(* Logix 5000 project; controller Transcat vendor 1 type 14 code 152 rev 32.11; software revision 32.02; part 2 of 2 *)
(* tags used below, declared in another part *)
   SpeedSensorUpperHowesSpeed : REAL;
   alwaysOFF : BOOL;
   FT103 : BronkhorstFlowMeter;
   FT104 : BronkhorstFlowMeter;
   FT105 : BronkhorstFlowMeter;
   GF101 : Thayer_WB_Feeder;   // Thayer 1 Tags
   GF201 : Thayer_WB_Feeder;   // Thayer 2 Tags
   GF301 : Acrison_Feeder;   // GF103 - Small Feeder 1
   MSG_FROM_SLC500 : INT[10];
   MX101 : Howes_Mixer;
   MX201 : Howes_Mixer;
   RecipeStart : BOOL;   // Bit to start and stop a recipe execution
   UpperHowesSpeed : INT;
   VF101 : Acrison_Feeder;   // Medium Feeder Tags
   VF201 : Acrison_Feeder;   // Small Feeder 2 Tags
(* MainProgram, continued *)

ROUTINE MainRoutine   (* ladder *)
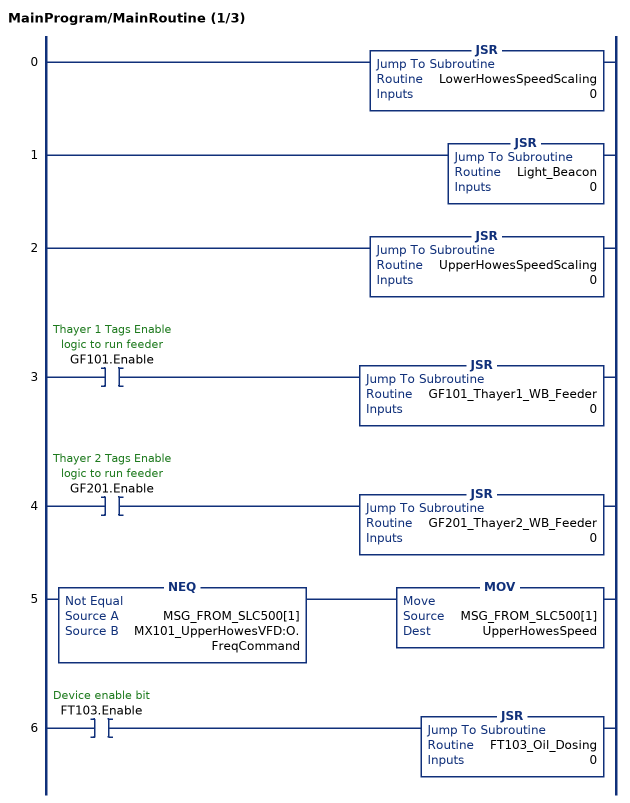
   0: JSR(LowerHowesSpeedScaling,0);
   1: JSR(Light_Beacon,0);
   2: JSR(UpperHowesSpeedScaling,0);
   3: XIC(GF101.Enable)JSR(GF101_Thayer1_WB_Feeder,0);
   4: XIC(GF201.Enable)JSR(GF201_Thayer2_WB_Feeder,0);
   5: NEQ(MSG_FROM_SLC500[1],MX101_UpperHowesVFD:O.FreqCommand)MOV(MSG_FROM_SLC500[1],UpperHowesSpeed);
   6: XIC(FT103.Enable)JSR(FT103_Oil_Dosing,0);
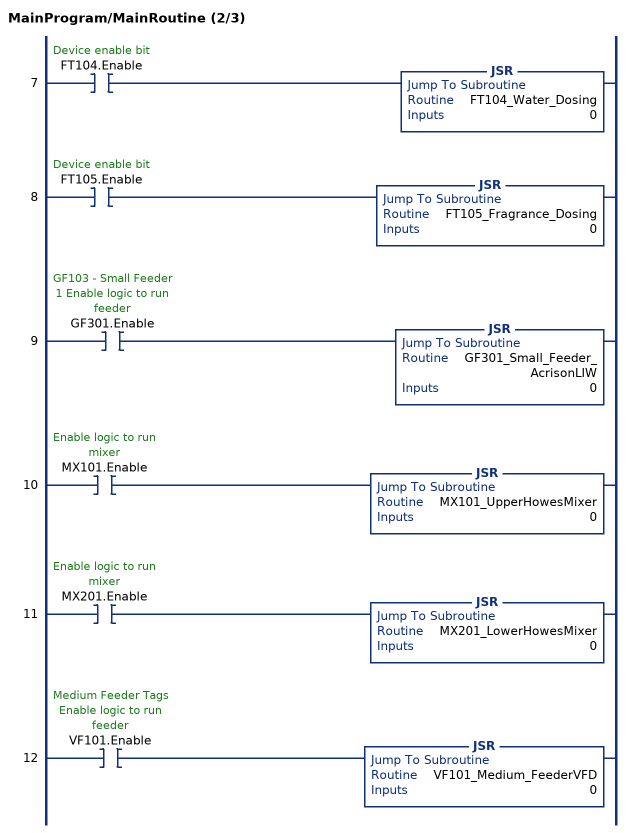
   7: XIC(FT104.Enable)JSR(FT104_Water_Dosing,0);
   8: XIC(FT105.Enable)JSR(FT105_Fragrance_Dosing,0);
   9: XIC(GF301.Enable)JSR(GF301_Small_Feeder_AcrisonLIW,0);
   10: XIC(MX101.Enable)JSR(MX101_UpperHowesMixer,0);
   11: XIC(MX201.Enable)JSR(MX201_LowerHowesMixer,0);
   12: XIC(VF101.Enable)JSR(VF101_Medium_FeederVFD,0);
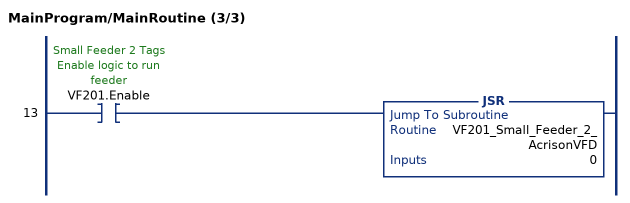
   13: XIC(VF201.Enable)JSR(VF201_Small_Feeder_2_AcrisonVFD,0);
END_ROUTINE

ROUTINE MX101_UpperHowesMixer   (* ladder *)
// Upper Howes Mixer Control Logic
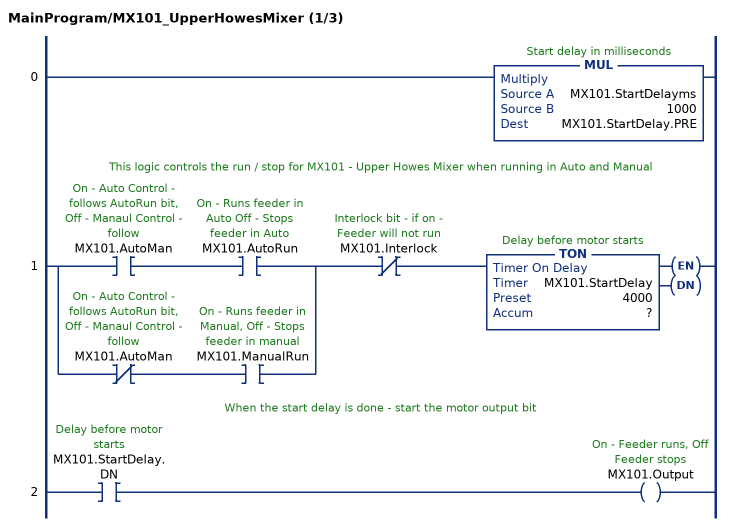
   0: MUL(MX101.StartDelayms,1000,MX101.StartDelay.PRE);
   // This logic controls the run / stop for MX101 - Upper Howes Mixer when running in Auto and Manual
   1: [XIC(MX101.AutoMan) XIC(MX101.AutoRun) ,XIO(MX101.AutoMan) XIC(MX101.ManualRun) ]XIO(MX101.Interlock)TON(MX101.StartDelay,?,?);
   // When the start delay is done - start the motor output bit
   2: XIC(MX101.StartDelay.DN)OTE(MX101.Output);
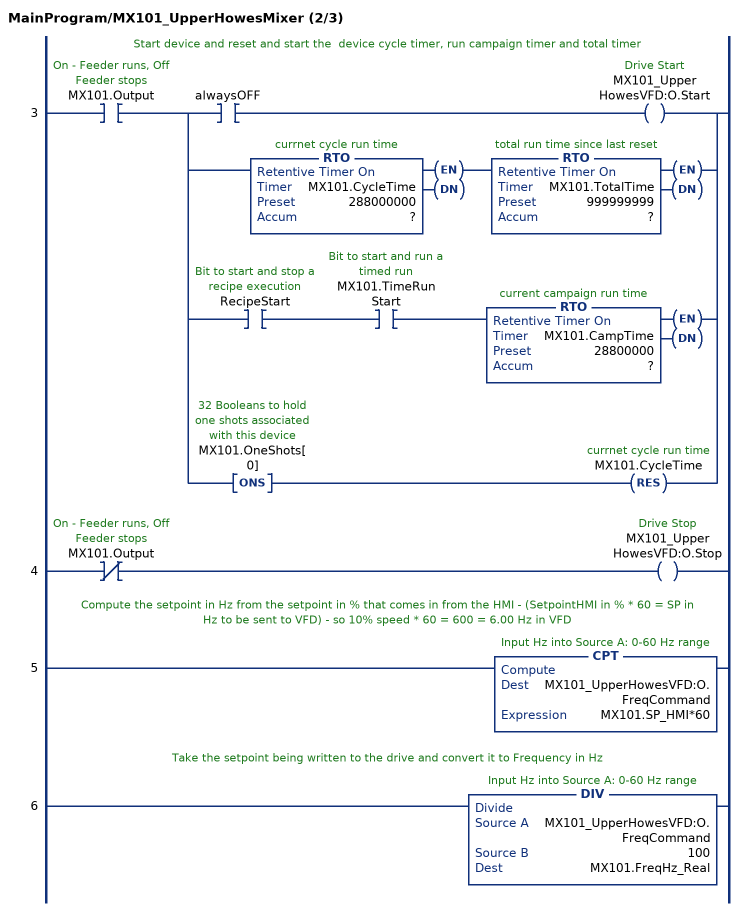
   // Start device and reset and start the  device cycle timer, run campaign timer and total timer
   3: XIC(MX101.Output)[XIC(alwaysOFF) OTE(MX101_UpperHowesVFD:O.Start) ,[RTO(MX101.CycleTime,?,?) RTO(MX101.TotalTime,?,?) ,XIC(RecipeStart) XIC(MX101.TimeRunStart) RTO(MX101.CampTime,?,?) ,ONS(MX101.OneShots[0]) RES(MX101.CycleTime) ] ];
   4: XIO(MX101.Output)OTE(MX101_UpperHowesVFD:O.Stop);
   // Compute the setpoint in Hz from the setpoint in % that comes in from the HMI - (SetpointHMI in % * 60 = SP in Hz to be sent to VFD) - so 10% speed * 60 = 600 = 6.00 Hz in VFD
   5: CPT(MX101_UpperHowesVFD:O.FreqCommand,MX101.SP_HMI*60);
   // Take the setpoint being written to the drive and convert it to Frequency in Hz
   6: DIV(MX101_UpperHowesVFD:O.FreqCommand,100,MX101.FreqHz_Real);
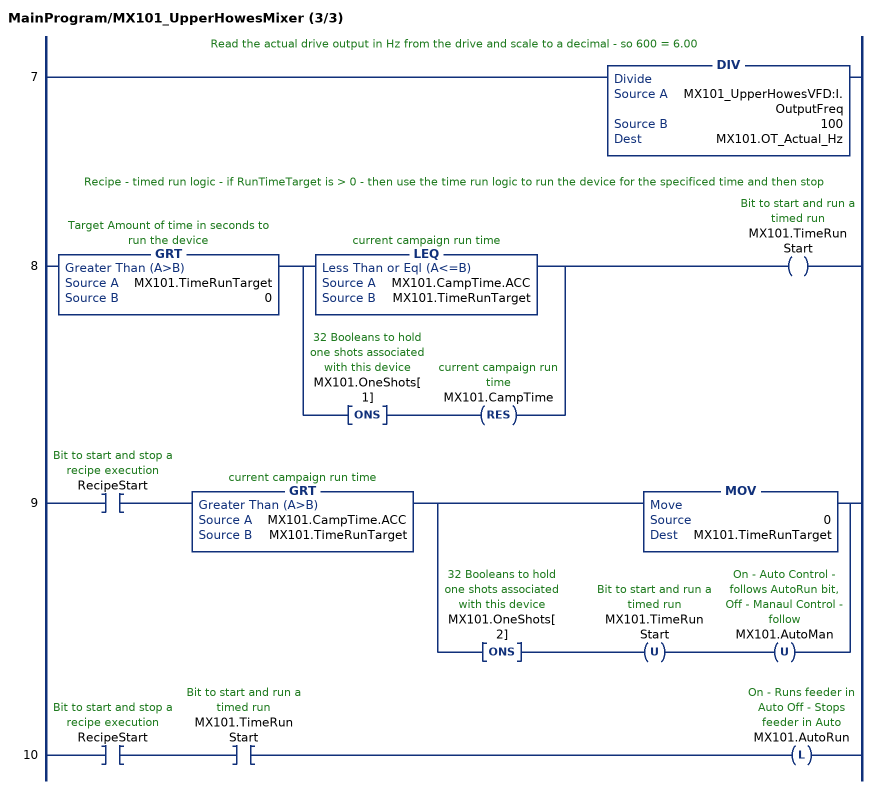
   // Read the actual drive output in Hz from the drive and scale to a decimal - so 600 = 6.00
   7: DIV(MX101_UpperHowesVFD:I.OutputFreq,100,MX101.OT_Actual_Hz);
   // Recipe - timed run logic - if RunTimeTarget is > 0 - then use the time run logic to run the device for the specificed time and then stop
   8: GRT(MX101.TimeRunTarget,0)[LEQ(MX101.CampTime.ACC,MX101.TimeRunTarget) ,ONS(MX101.OneShots[1]) RES(MX101.CampTime) ]OTE(MX101.TimeRunStart);
   9: XIC(RecipeStart)GRT(MX101.CampTime.ACC,MX101.TimeRunTarget)[MOV(0,MX101.TimeRunTarget) ,ONS(MX101.OneShots[2]) OTU(MX101.TimeRunStart) OTU(MX101.AutoMan) ];
   10: XIC(RecipeStart)XIC(MX101.TimeRunStart)OTL(MX101.AutoRun);
END_ROUTINE

ROUTINE MX201_LowerHowesMixer   (* ladder *)
// Lower Howes Mixer Control Logic
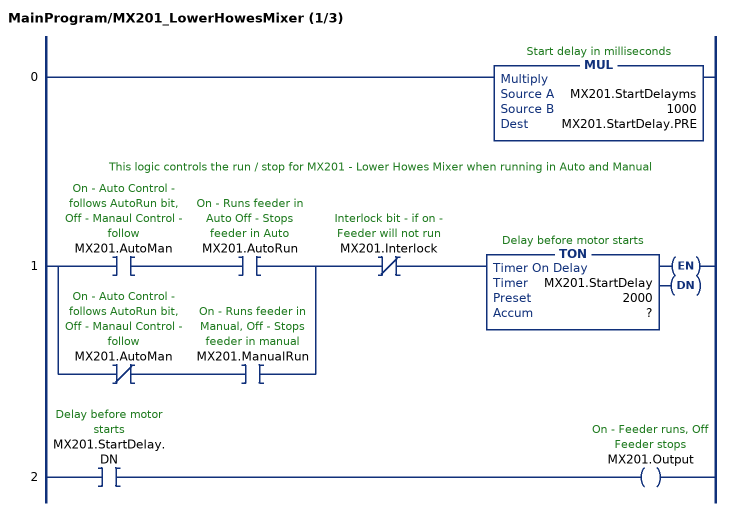
   0: MUL(MX201.StartDelayms,1000,MX201.StartDelay.PRE);
   // This logic controls the run / stop for MX201 - Lower Howes Mixer when running in Auto and Manual
   1: [XIC(MX201.AutoMan) XIC(MX201.AutoRun) ,XIO(MX201.AutoMan) XIC(MX201.ManualRun) ]XIO(MX201.Interlock)TON(MX201.StartDelay,?,?);
   2: XIC(MX201.StartDelay.DN)OTE(MX201.Output);
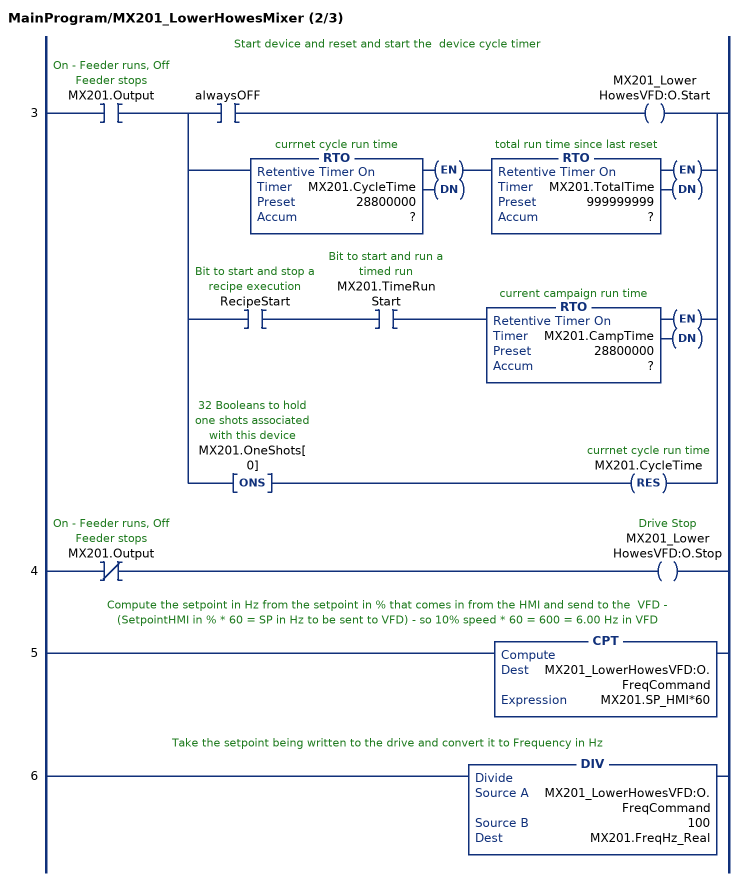
   // Start device and reset and start the  device cycle timer
   3: XIC(MX201.Output)[XIC(alwaysOFF) OTE(MX201_LowerHowesVFD:O.Start) ,[[RTO(MX201.CycleTime,?,?) RTO(MX201.TotalTime,?,?) ,XIC(RecipeStart) XIC(MX201.TimeRunStart) RTO(MX201.CampTime,?,?) ] ,ONS(MX201.OneShots[0]) RES(MX201.CycleTime) ] ];
   4: XIO(MX201.Output)OTE(MX201_LowerHowesVFD:O.Stop);
   // Compute the setpoint in Hz from the setpoint in % that comes in from the HMI and send to the  VFD - (SetpointHMI in % * 60 = SP in Hz to be sent to VFD) - so 10% speed * 60 = 600 = 6.00 Hz in VFD
   5: CPT(MX201_LowerHowesVFD:O.FreqCommand,MX201.SP_HMI*60);
   // Take the setpoint being written to the drive and convert it to Frequency in Hz
   6: DIV(MX201_LowerHowesVFD:O.FreqCommand,100,MX201.FreqHz_Real);
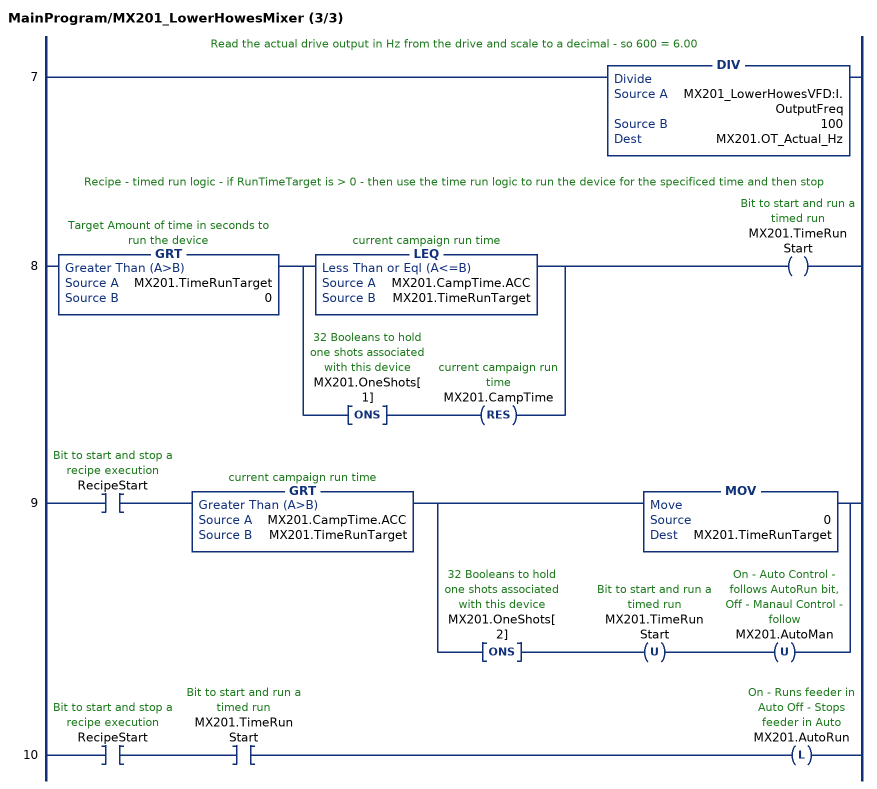
   // Read the actual drive output in Hz from the drive and scale to a decimal - so 600 = 6.00
   7: DIV(MX201_LowerHowesVFD:I.OutputFreq,100,MX201.OT_Actual_Hz);
   // Recipe - timed run logic - if RunTimeTarget is > 0 - then use the time run logic to run the device for the specificed time and then stop
   8: GRT(MX201.TimeRunTarget,0)[LEQ(MX201.CampTime.ACC,MX201.TimeRunTarget) ,ONS(MX201.OneShots[1]) RES(MX201.CampTime) ]OTE(MX201.TimeRunStart);
   9: XIC(RecipeStart)GRT(MX201.CampTime.ACC,MX201.TimeRunTarget)[MOV(0,MX201.TimeRunTarget) ,ONS(MX201.OneShots[2]) OTU(MX201.TimeRunStart) OTU(MX201.AutoMan) ];
   10: XIC(RecipeStart)XIC(MX201.TimeRunStart)OTL(MX201.AutoRun);
END_ROUTINE

ROUTINE UpperHowesSpeedScaling   (* function block diagram *)
// 4-20 MillAmp scaling
   SHEET 1
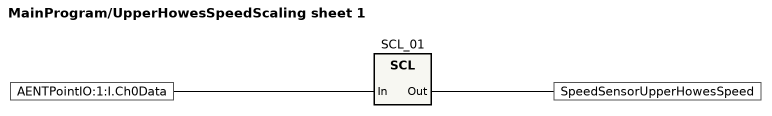
   SCL_01 : SCL(In := AENTPointIO:1:I.Ch0Data);
   SpeedSensorUpperHowesSpeed := SCL_01.Out;
END_ROUTINE

ROUTINE VF101_Medium_FeederVFD   (* ladder *)
// Medium Feeder Control via PowerFlex 525 VFD
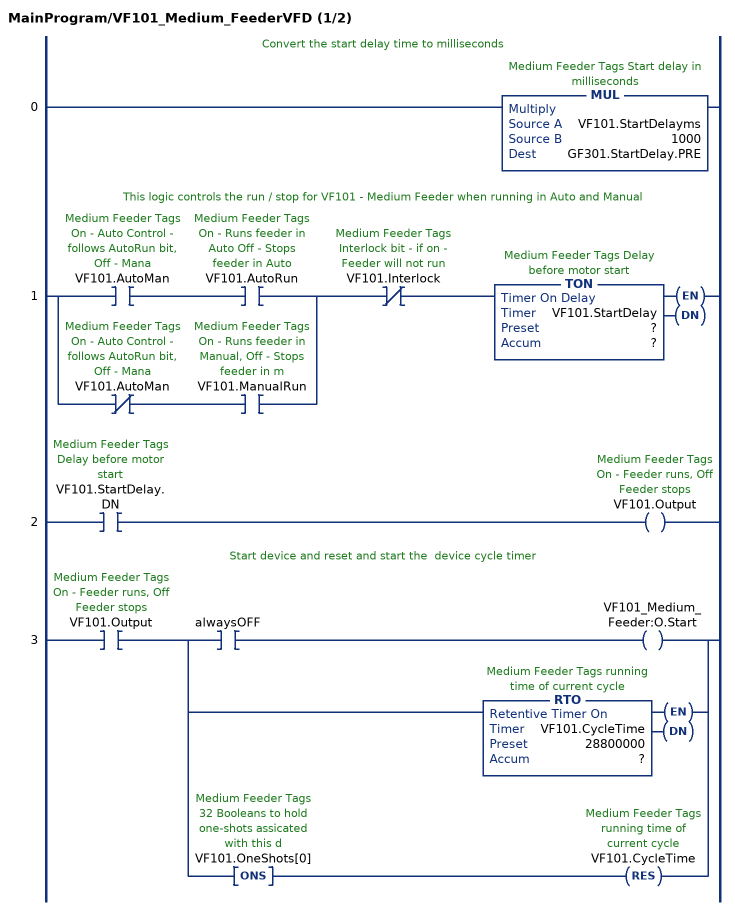
   // Convert the start delay time to milliseconds
   0: MUL(VF101.StartDelayms,1000,GF301.StartDelay.PRE);
   // This logic controls the run / stop for VF101 - Medium Feeder when running in Auto and Manual
   1: [XIC(VF101.AutoMan) XIC(VF101.AutoRun) ,XIO(VF101.AutoMan) XIC(VF101.ManualRun) ]XIO(VF101.Interlock)TON(VF101.StartDelay,?,?);
   2: XIC(VF101.StartDelay.DN)OTE(VF101.Output);
   // Start device and reset and start the  device cycle timer
   3: XIC(VF101.Output)[XIC(alwaysOFF) OTE(VF101_Medium_Feeder:O.Start) ,[RTO(VF101.CycleTime,?,?) ,ONS(VF101.OneShots[0]) RES(VF101.CycleTime) ] ];
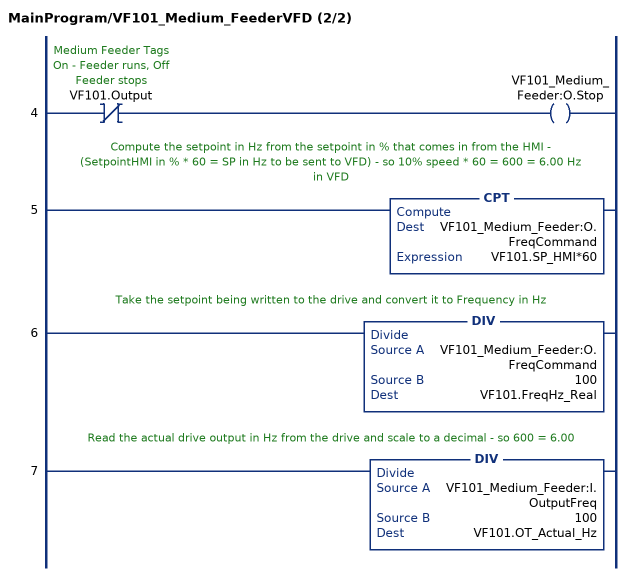
   4: XIO(VF101.Output)OTE(VF101_Medium_Feeder:O.Stop);
   // Compute the setpoint in Hz from the setpoint in % that comes in from the HMI - (SetpointHMI in % * 60 = SP in Hz to be sent to VFD) - so 10% speed * 60 = 600 = 6.00 Hz in VFD
   5: CPT(VF101_Medium_Feeder:O.FreqCommand,VF101.SP_HMI*60);
   // Take the setpoint being written to the drive and convert it to Frequency in Hz
   6: DIV(VF101_Medium_Feeder:O.FreqCommand,100,VF101.FreqHz_Real);
   // Read the actual drive output in Hz from the drive and scale to a decimal - so 600 = 6.00
   7: DIV(VF101_Medium_Feeder:I.OutputFreq,100,VF101.OT_Actual_Hz);
END_ROUTINE

ROUTINE VF201_Small_Feeder_2_AcrisonVFD   (* ladder *)
// Small Feeder 2 - Control via PowerFlex 525 VFD
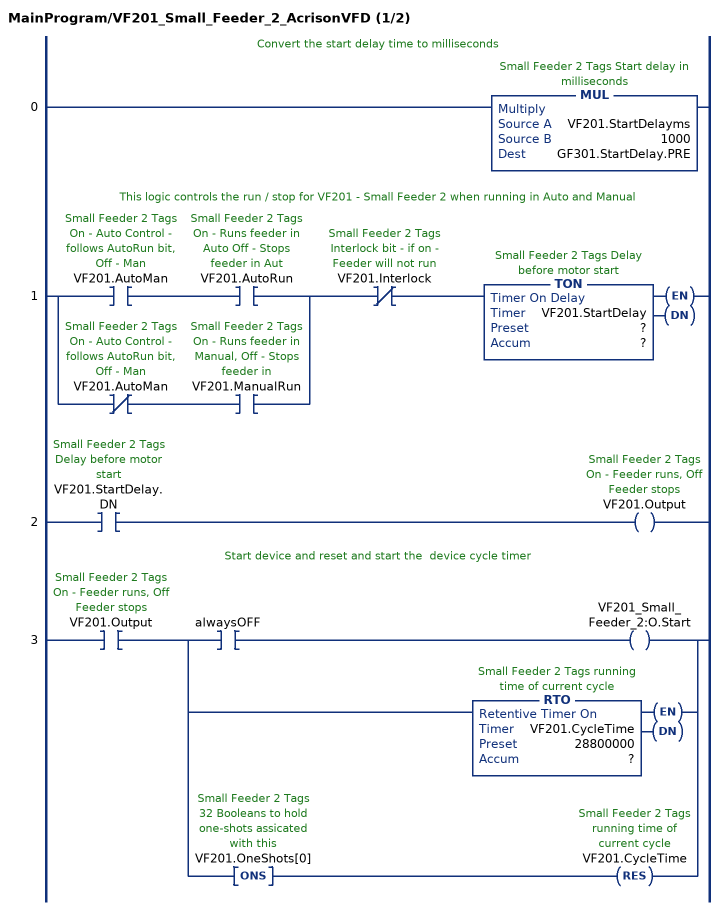
   // Convert the start delay time to milliseconds
   0: MUL(VF201.StartDelayms,1000,GF301.StartDelay.PRE);
   // This logic controls the run / stop for VF201 - Small Feeder 2 when running in Auto and Manual
   1: [XIC(VF201.AutoMan) XIC(VF201.AutoRun) ,XIO(VF201.AutoMan) XIC(VF201.ManualRun) ]XIO(VF201.Interlock)TON(VF201.StartDelay,?,?);
   2: XIC(VF201.StartDelay.DN)OTE(VF201.Output);
   // Start device and reset and start the  device cycle timer
   3: XIC(VF201.Output)[XIC(alwaysOFF) OTE(VF201_Small_Feeder_2:O.Start) ,[RTO(VF201.CycleTime,?,?) ,ONS(VF201.OneShots[0]) RES(VF201.CycleTime) ] ];
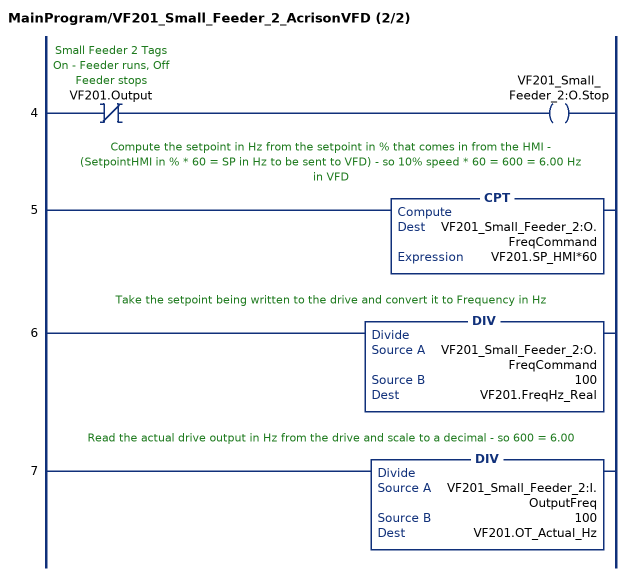
   4: XIO(VF201.Output)OTE(VF201_Small_Feeder_2:O.Stop);
   // Compute the setpoint in Hz from the setpoint in % that comes in from the HMI - (SetpointHMI in % * 60 = SP in Hz to be sent to VFD) - so 10% speed * 60 = 600 = 6.00 Hz in VFD
   5: CPT(VF201_Small_Feeder_2:O.FreqCommand,VF201.SP_HMI*60);
   // Take the setpoint being written to the drive and convert it to Frequency in Hz
   6: DIV(VF201_Small_Feeder_2:O.FreqCommand,100,VF201.FreqHz_Real);
   // Read the actual drive output in Hz from the drive and scale to a decimal - so 600 = 6.00
   7: DIV(VF201_Small_Feeder_2:I.OutputFreq,100,VF201.OT_Actual_Hz);
END_ROUTINE
END_PROGRAM
